FUNCTION_BLOCK PVActor (* Actor for sending data to the PhotovoltaicsActor plugin controller in Polysun. *)
  (* Standard: 61499-2 *)
  (* Version 1.0, 2017-07-21, Marc Jakobi, HTW Berlin *)
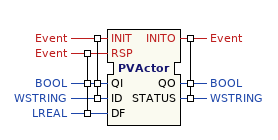
  EVENT_INPUT
    INIT WITH QI, ID; (* Service Initialization *)
    RSP WITH DF, QI; (* Service Response *)
  END_EVENT
  EVENT_OUTPUT
    INITO WITH QO, STATUS; (* Initialization Confirm *)
  END_EVENT
  VAR_INPUT
    QI : BOOL; (* Input event qualifier *)
    ID : WSTRING; (* Connection Identifier *)
    DF : LREAL; (* Derating factor  [0,..,1] *)
  END_VAR
  VAR_OUTPUT
    QO : BOOL; (* Output event qualifier *)
    STATUS : WSTRING; (* Service status *)
  END_VAR
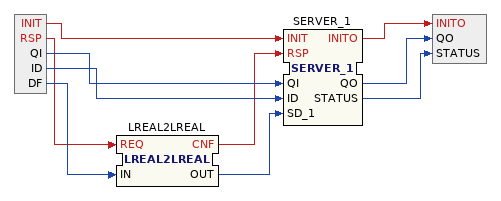
  FBS
    SERVER_1 : SERVER_1;
    LREAL2LREAL : LREAL2LREAL;
  END_FBS
  EVENT_CONNECTIONS
    INIT TO SERVER_1.INIT;
    SERVER_1.INITO TO INITO;
    RSP TO LREAL2LREAL.REQ;
    LREAL2LREAL.CNF TO SERVER_1.RSP;
  END_CONNECTIONS
  DATA_CONNECTIONS
    QI TO SERVER_1.QI;
    ID TO SERVER_1.ID;
    SERVER_1.QO TO QO;
    SERVER_1.STATUS TO STATUS;
    DF TO LREAL2LREAL.IN;
    LREAL2LREAL.OUT TO SERVER_1.SD_1;
  END_CONNECTIONS
END_FUNCTION_BLOCK
